FUNCTION_BLOCK ADD_DT_TIME (* IEC 61131-3 DATE_AND_TIME+TIME *)
  (* Standard: 61131-3 *)
  (* Version 0.0, 2004-12-15, JHC, Rockwell Automation, Converted from SRC format. *)
  (* Compiler header: package fb.rt.plc.math; *)
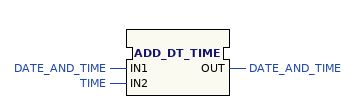
  VAR_INPUT
    IN1 : DATE_AND_TIME; (* Augend *)
    IN2 : TIME; (* Addend *)
  END_VAR
  VAR_OUTPUT
    OUT : DATE_AND_TIME; (* Sum *)
  END_VAR
END_FUNCTION_BLOCK
